// TIA Portal V16 export
// export: Created 2025-10-06T17:54:29.6304535Z, ExportSetting WithDefaults, DisplayName Totally Integrated Automation Portal, DisplayVersion V16, DisplayName TIA Portal Version Control Interface, DisplayVersion V16, DisplayName TIA Portal Openness, DisplayVersion V16, DisplayName STEP 7 Professional, DisplayVersion V16, DisplayName STEP 7 Safety, DisplayVersion V16, DisplayName WinCC Advanced, DisplayVersion V16
FUNCTION_BLOCK "Override_Block_Safety"   // FB7, FBD
TITLE = Override Block Safety.
VERSION : 0.1
// stored: AutoNumber true, IsIECCheckEnabled false, UDAEnableTagReadback false
   VAR_INPUT
      "SAFE Q 1" : Bool;
      "SAFE Q 2" : Bool;
      "Override Contact" : Bool;
      "Delay Timer" : Time;
   END_VAR
   VAR_OUTPUT
      "SAFE Output Contact" : Bool;
      "Timer ET" : Time;
   END_VAR
BEGIN

REGION Network 1: SAFETY - OVERRIDE
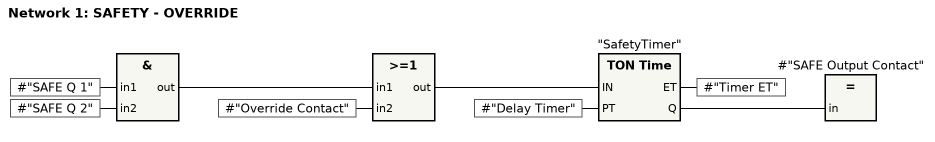
   "SafetyTimer".TON(IN := (#"SAFE Q 1" AND #"SAFE Q 2") OR #"Override Contact",
                     PT := #"Delay Timer",
                     ET => #"Timer ET");
   #"SAFE Output Contact" := "SafetyTimer".Q;
END_REGION
END_FUNCTION_BLOCK
